{attribute 'linkalways'} 
{attribute 'no_explicit_call' := 'This FB is a CLASS and must be accessed using methods or properties'}
{attribute 'enable_dynamic_creation'}
FUNCTION_BLOCK FINAL MOD_UDINT EXTENDS Node
VAR
	in1 : _UDINT(0);
	in2 : _UDINT(0);
	out : _UDINT(0);
END_VAR

METHOD PUBLIC Clone : I_Node
VAR
	pNode : POINTER TO MOD_UDINT;
END_VAR
pNode := __NEW(MOD_UDINT);
Clone := pNode^;
END_METHOD

METHOD FB_init : BOOL
VAR_INPUT
	bInitRetains : BOOL; // if TRUE, the retain variables are initialized (warm start / cold start)
	bInCopyCode : BOOL;  // if TRUE, the instance afterwards gets moved into the copy code (online change)
END_VAR
AddInput('in1',THIS^.in1);
AddInput('in2',THIS^.in2);
AddOutput('out', THIS^.out);
END_METHOD

METHOD PROTECTED OnExecute
VAR
END_VAR
out.Value := in1.Value MOD in2.Value;
END_METHOD

END_FUNCTION_BLOCK

(* stored: Version 1.1.0.1, ProductVersion 3.1.4024.15
   POU MOD_UDINT: Id {76ffd789-1304-4a09-8550-7d627d173553}, SpecialFunc None
   Folder Constructor: Id {4a1a60b6-0a79-431a-81cd-9ccacedf44c9}
   Method Clone: Id {40680dba-543d-444a-908d-f1319df0f085}
   Method FB_init: Id {4cd7dcb1-6e3e-470a-8307-857a50938f16}
   Method OnExecute: Id {af38322e-23c0-4cc0-a57f-baf0f8e843d4} *)
